(* IEC 61131-3 sources: RL_MAR/experiments/comparison/llm4plc/results/gpt-4o-mini_20260506_100619/20260506_102652, 1 file *)

(* ---- generated_code_iteration_0.st ---- *)
ructured-text
START_ST
FUNCTION_BLOCK TrafficManagementSystem
    VAR_INPUT
        VehicleCount1 : INT; // Vehicle count at intersection 1
        VehicleCount2 : INT; // Vehicle count at intersection 2
        VehicleCount3 : INT; // Vehicle count at intersection 3
        VehicleCount4 : INT; // Vehicle count at intersection 4
    END_VAR

    VAR_OUTPUT
        TrafficLight1 : BOOL; // Traffic light state for intersection 1
        TrafficLight2 : BOOL; // Traffic light state for intersection 2
        TrafficLight3 : BOOL; // Traffic light state for intersection 3
        TrafficLight4 : BOOL; // Traffic light state for intersection 4
    END_VAR

    VAR
        state: INT; // Current state of the FSM
        prevState: INT; // Previous state variable
    END_VAR

    // Initialize the state
    state := 0;
    TrafficLight1 := FALSE;
    TrafficLight2 := FALSE;
    TrafficLight3 := FALSE;
    TrafficLight4 := FALSE;

    // State machine logic
    CASE state OF
        0: // STATE 0: INITIALIZE
            TrafficLight1 := FALSE;
            TrafficLight2 := FALSE;
            TrafficLight3 := FALSE;
            TrafficLight4 := FALSE;
            state := 1; // Transition to STATE 1

        1: // STATE 1: SET TRAFFIC LIGHTS FOR INTERSECTION 1 AND 2
            IF VehicleCount1 > VehicleCount2 THEN
                TrafficLight1 := TRUE;
                TrafficLight2 := FALSE;
            ELSE
                TrafficLight1 := FALSE;
                TrafficLight2 := TRUE;
            END_IF;
            state := 2; // Transition to STATE 2

        2: // STATE 2: SET TRAFFIC LIGHTS FOR INTERSECTION 3 AND 4
            IF VehicleCount3 > VehicleCount4 THEN
                TrafficLight3 := TRUE;
                TrafficLight4 := FALSE;
            ELSE
                TrafficLight3 := FALSE;
                TrafficLight4 := TRUE;
            END_IF;
            state := 1; // Transition back to STATE 1
    END_CASE

END_FUNCTION_BLOCK
END_ST
